PROGRAM MAIN
VAR
	fbEL6021RTD				: FB_SerialCom;
	fbEL6021TC				: FB_SerialCom;
	fbEL6002Flow			: FB_SerialCom;
	fbEL6021_MB				: FB_SerialCom;
	fbDoesItWork			: FB_SanityCheck;
	fbFormatRTD				: FB_FormatTempRTD;
	fbFormatTC				: FB_FormatTempTC;
	fbmVtoTemp				: FB_mVtoTemp;
	fbLedOff				: FB_LedOff;
	error					: ComError_t;
	fbPID					: FB_Ploop;
//	fbCloseValve1			: FB_CloseValve;
	fbMoveAxis1Rel			: FB_MoveStepperRel;
	fbMoveAxis1Abs			: FB_MoveStepperAbs;
	fbStepperLoop			: FB_MoveStepperLoop;
	
// Modbus Fan Control Variables
	Fan1 					: FB_FanModbus; // FB for controlling Ebm Pabst Fan over Modbus
	fbCCMT4mb				: FB_ValveModbus;
	fbSetupCCMTmb			: FB_CCMT4Setup;
	bFanEnable				: BOOL;
	mbReadAddr				: WORD := 16#D000;
	mbWriteAddr 			: WORD := 16#D000;
	mbReadData				: WORD;
	mbWriteData 			: WORD;
	smbRPM					: STRING;
	mbRPM					: WORD;
	tachometerData 			: REAL;
	speedNominal 			: REAL;
	
// Stepper Variables
	bJogFwd					: BOOL;
	bJogBack				: BOOL;
	bJogDone				: BOOL;
	bValve1Closed			: BOOL;

// Modbus Valve Variables
	percentOD				: STRING;
	cmdOD					: REAL;
	btnMbActivate 			: BOOL := FALSE;
	ccmtPos					: WORD;
	sCCMTPos				: STRING;
	bSetupComplete			: BOOL := 0;

// Misc. Variables	
	sVaporQual				: STRING;
	sTemp01					: STRING;
	sTemp02					: STRING;
	sPress01				: STRING;
	sPress02				: STRING;
	sPress03				: STRING;
	sPress04				: STRING;
	SurfaceRTD1 			: STRING;
	SurfaceRTD2 			: STRING;
	sStepperGoTo			: STRING;
	sStepperNumSteps		: STRING;
	RTDorTC					: BOOL;
	
	bTest					: BOOL := FALSE;
	TEST					: BOOL := FALSE;

///////////////////////////////////////////////////////////////////////
//Function16
	_MBWriteRegs	:FB_MBWriteRegs;
	MBWriteRegs		:DUT_MB;
	ar2				:ARRAY[0..99] OF INT;
	
	//Function3
	_MBReadRegs		:FB_ModBusTCPReadRegs;
	MBReadRegs		:DUT_MBReads;
	ar1				:ARRAY[0..99] OF INT;
	
	sIPAddr:STRING(15):='192.168.000.001';



END_VAR
VAR_INPUT
	fbAxis1					: FB_StepperCtrl;
	fbAxis2					: FB_StepperCtrl;
	msgOutRTD				: STRING;
	msgOutTC				: STRING;
	msgOutFlow				: STRING;
	TempRaw					: STRING;
	MoveTo					: UDINT;
	StepsToMove				: UDINT;
	bMoveRelative			: BOOL := FALSE;
	bMoveAbsolute			: BOOL := FALSE;
END_VAR
VAR_OUTPUT
	bDirection				: BOOL;
END_VAR

///////////////////////////////////////////
// CLOSE VALVES ON STARTUP
///////////////////////////////////////////
//WHILE bValve1Closed <> TRUE DO
//	fbCloseValve1(bDone => bValve1Closed); 
//END_WHILE

// CCMT 4 Modbus Setup Routine
IF bSetupComplete = 0 THEN
	fbSetupCCMTmb(bSetupComplete => bSetupComplete);
END_IF


///////////////////////////////////////////
// CALL RS-485 ROUTINE
///////////////////////////////////////////
Background();

///////////////////////////////////////////
// RTD AND TC TEMP READINGS
///////////////////////////////////////////

fbEL6021RTD(
	TxBuffer := TxBufferEL_RTD,
	RxBuffer := RxBufferEL_RTD,
	msgOUT => msgOutRTD,
	prefix := '°C',
	suffix := ','
);

fbFormatRTD(
	sTempRaw := msgOutRTD, 
);
	
fbEL6021TC(
	TxBuffer := TxBufferEL_TC,
	RxBuffer := RxBufferEL_TC,
	msgOUT => msgOutTC,
	prefix := 'mV',
	suffix := ','
);
	
fbFormatTC(
	sTempRaw := msgOutTC
);

fbmVtoTemp(mVtempArray := fbFormatTC.tempArray);
fbmVtoTemp(T_cj := (INT_TO_LREAL(GVL.RTD4Ch1) / 10));

///////////////////////////////////////////
// FLOW METER RS-232
///////////////////////////////////////////

fbEL6002Flow(
	TxBuffer := TxBufferEL_Flow,
	RxBuffer := RxBufferEL_Flow,
	msgOUT => msgOutFlow,
	prefix := ,//'$N',
	suffix := //'$R'
);

///////////////////////////////////////////
// CALL BLINKENLIGHTS SANITY CHECK
///////////////////////////////////////////
fbDoesItWork();

///////////////////////////////////////////
// CALL VALVE PID CONTROL
///////////////////////////////////////////
fbPID(
		fSetPointValue := 100
);

///////////////////////////////////////////
// FORMAT AHU BOARD DATA FOR GUI
///////////////////////////////////////////
sVaporQual := TO_STRING(20 - 16 * (INT_TO_REAL(GVL.aiHBX01) / 32767));
sPress01 := TO_STRING(100 * (INT_TO_REAL((GVL.aiPress01) * 2) / 65536));
sPress02 := TO_STRING(100 * (INT_TO_REAL((GVL.aiPress02) * 2) / 65536));
sPress03 := TO_STRING(100 * (INT_TO_REAL((GVL.aiPress03) * 2) / 65536));
sPress04 := TO_STRING(100 * (INT_TO_REAL((GVL.aiPress04) * 2) / 65536));
SurfaceRTD1 := TO_STRING(INT_TO_REAL(GVL.RTD2Ch1) / 10);
SurfaceRTD2 := TO_STRING(INT_TO_REAL(GVL.RTD2Ch2) / 10);

IF bJogFwd = TRUE THEN
	fbAxis1(bJogFwd := TRUE, bJogBack := FALSE, bJogDone => bJogDone);
END_IF

IF bJogBack = TRUE THEN
	fbAxis1(bJogBack := TRUE, bJogFwd := FALSE, bJogDone => bJogDone);
END_IF

IF (bJogFwd = FALSE AND bJogBack = FALSE) OR bJogDone = TRUE THEN
	fbAxis1(bJogFwd := FALSE, bJogBack := FALSE);
END_IF

IF bMoveRelative = TRUE THEN
	fbMoveAxis1Rel(
		stepsToMove := STRING_TO_INT(sStepperNumSteps)
	);
END_IF

IF bMoveAbsolute = TRUE THEN
	fbMoveAxis1Abs(
		stepsToMove := STRING_TO_INT(sStepperGoTo)
	);
END_IF

IF TEST = TRUE THEN
	fbStepperLoop(
		stepsToMove := STRING_TO_INT(sStepperGoTo)
	);
END_IF

///////////////////////////////////////////
// FAN CONTROL
///////////////////////////////////////////


IF bFanEnable = TRUE THEN
	Fan1(
	f_mbReadAddr := mbReadAddr,
	f_mbWriteAddr := mbWriteAddr,
	f_mbWriteData := mbWriteData,
	f_mbRPM := TO_WORD(smbRPM),
	//f_state := state,
	//f_nextState := nextState,
	f_mbReadData => mbReadData,
	f_tachometerData => tachometerData,
	f_speedNominal => speedNominal
);
ELSE
	Fan1(
	f_mbReadAddr := mbReadAddr,
	f_mbWriteAddr := mbWriteAddr,
	f_mbWriteData := mbWriteData,
	f_mbRPM := 0,
	//f_state := state,
	//f_nextState := nextState,
	f_mbReadData => mbReadData,
	f_tachometerData => tachometerData,
	f_speedNominal => speedNominal
);
END_IF

// CCMT 4 Modbus Control

cmdOD := ((STRING_TO_REAL(percentOD) / 1100) * 1000);
IF STRING_TO_REAL(percentOD) > 1100 THEN
	percentOD := '1100';
END_IF
IF cmdOD > 1000 THEN
	cmdOD := 1000;
END_IF
IF cmdOD < 0 THEN
	cmdOD := 0;
END_IF

IF btnMbActivate = TRUE THEN
	fbCCMT4mb(
		posData := REAL_TO_WORD(cmdOD),
		posActualData => ccmtPos
		);
		sCCMTPos := WORD_TO_STRING(ccmtPos);
ELSE
	fbCCMT4mb(
		posData := 0,
		posActualData => ccmtPos
		);
		sCCMTPos := WORD_TO_STRING(ccmtPos);
END_IF

fbLedOff();
fbEL6021_MB(
	RxBuffer := GVL.RxBufferEL_MB, 
	TxBuffer := GVL.TxBufferEL_MB
);

END_PROGRAM

(* stored: Version 1.1.0.1, ProductVersion 3.1.4026.7
   POU MAIN: Id {dd0522d0-2de6-4616-8ca5-ff1eaf6afbeb}, SpecialFunc None *)
